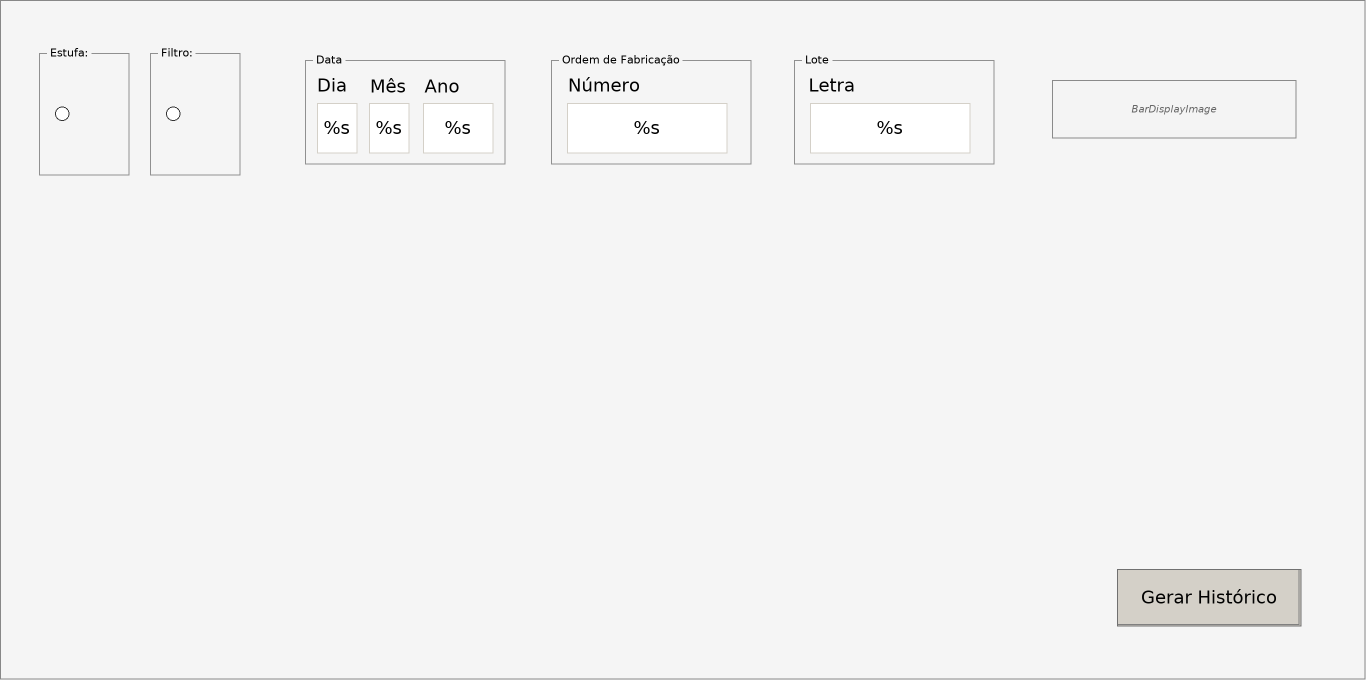
VISUALIZATION Historical  // 1366x680
    GroupBox (39,45 90x130), "Estufa:"
        RadioButton (14,24 65x89), variable: GVL.radioEstufa
            Areas[0]: Text=019
            Areas[1]: Text=020
            Areas[2]: Text=021
    Textfield (317,103 40x50), "%s", text variable: GVL.arrCVSfilter[GVL.radioEstufa].dia, input disabled if: GVL.radioData
        OnMouseClick: write the text variable via VisuDialogs.Numpad
    GroupBox (150,45 90x130), "Filtro:"
        RadioButton (14,24 65x89), variable: GVL.radioFiltro
            Areas[0]: Text=Data
            Areas[2]: Text=Lote
    BarDisplayImage (1052,80 244x58), value: P_TextModeWrite.nRow, style: BarDisplayImage-Gray, scale format: %.1f, scale 0..100
        p518627256: Gerando ...
    Textfield (369,103 40x50), "%s", text variable: GVL.arrCVSfilter[GVL.radioEstufa].mes, input disabled if: GVL.radioData
        OnMouseClick: write the text variable via VisuDialogs.Numpad
    Textfield (423,103 70x50), "%s", text variable: GVL.arrCVSfilter[GVL.radioEstufa].ano, input disabled if: GVL.radioData
        OnMouseClick: write the text variable via VisuDialogs.Numpad
    GroupBox (551,52 200x112), "Ordem de Fabricação", input disabled if: GVL.radioOF
        Textfield (16,51 160x50), "%s", text variable: GVL.arrCVSfilter[GVL.radioEstufa].ordem, input disabled if: GVL.radioOF
            OnMouseClick: write the text variable via VisuDialogs.Numpad
        Label (13,19 80x29), "Número"
    GroupBox (794,52 200x112), "Lote", input disabled if: GVL.radioLote
        Textfield (16,51 160x50), "%s", text variable: GVL.arrCVSfilter[GVL.radioEstufa].lote, input disabled if: GVL.radioLote
            OnMouseClick: write the text variable via VisuDialogs.Keypad
        Label (12,19 52x29), "Letra"
    GroupBox (305,52 200x112), "Data", input disabled if: GVL.radioData
        Label (-13,19 80x29), "Dia"
        Label (43,20 80x29), "Mês"
        Label (97,20 80x29), "Ano"
    Button (1117,569 184x57), "Gerar Histórico"
        OnMouseClick: execute { gvl.bHistory:=true; }
END_VISUALIZATION

(* stored: Version 1.1.0.1, ProductVersion 3.1.4024.12
   Visu Historical: Id {3e4f0589-6098-4e7c-a35a-5508c5aa1d43} *)
